(* PLC project Unnamed, Unknown Unnamed 1 *)
(* stored: creationDateTime 2026-02-02T16:28:11, modificationDateTime 2026-02-02T16:32:03 *)

PROGRAM program0
  VAR
    EStop AT %IX0.2 : BOOL;
    GuardClosed AT %IX0.4 : BOOL;
    RunPermit AT %M00 : BOOL;
  END_VAR

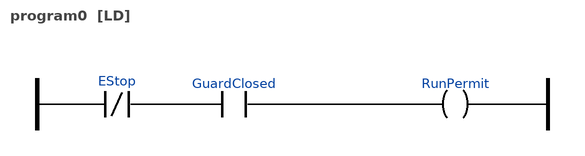
(* LD diagram, written out as Structured Text *)
RunPermit := NOT EStop AND GuardClosed;
END_PROGRAM

CONFIGURATION Config0
  RESOURCE Res0 ON PLC
    TASK task0(INTERVAL := T#20ms, PRIORITY := 0);
    PROGRAM instance0 WITH task0 : program0;
  END_RESOURCE
END_CONFIGURATION
